# EPICS autosave request: iocBoot/iocTomoScan_13BM_PSO/auto_settings.req
file "tomoScan_settings.req", P=$(P), R=$(R)
file "tomoScan_PSO_settings.req", P=$(P), R=$(R)
file "tomoScan_13BM_PSO_settings.req", P=$(P), R=$(R)
